PROGRAM PRG_VfdModbusRtu
VAR
	fbVfdMb: ModbusRtuMaster_KL6x22B;
	fbRTrigWrite: R_Trig;
	fbRTrigEnable: R_Trig;
	fbRTrigDisable: R_Trig;
	fbTON: TON;
	wQty: WORD := 1;
	wMbAddr: WORD;
	wCmd: WORD;
	bWrite: BOOL;
END_VAR

fbRTrigWrite(CLK:=bWrite, Q=>);
fbRTrigEnable(CLK:=GVL.bEnable, Q=>);
fbRTrigEnable(CLK:=GVL.bDisable, Q=>);

IF fbRTrigEnable.Q THEN
	bWrite := TRUE;
	fbTON(IN:= bWrite, PT:= T#500MS, Q=> , ET=> );
	wMbAddr := 416;
	wCmd := 1;
END_IF

IF fbRTrigDisable.Q THEN
	bWrite := TRUE;
	fbTON(IN:= bWrite, PT:= T#500MS, Q=> , ET=> );
	wMbAddr := 416;
	wCmd := 0;
END_IF

IF fbTON.Q THEN
	fbTON(IN:=FALSE);
	bWrite := FALSE;
END_IF

fbVfdMb.WriteRegs(
	UnitID:= 1, 
	Quantity:= wQty, 
	MBAddr:= wMbAddr, 
	cbLength:= SIZEOF(wCmd), 
	pMemoryAddr:= ADR(wCmd), 
	Execute:= fbRTrigWrite.Q, 
	Timeout:= T#1S, 
	BUSY=> , 
	Error=> , 
	ErrorId=> , 
	cbRead=> );

END_PROGRAM

(* stored: Version 1.1.0.1, ProductVersion 3.1.4024.12
   POU PRG_VfdModbusRtu: Id {9519abab-4381-406c-81bf-d5d84071b90e}, SpecialFunc None *)
